{attribute addProperty BoxType "AX5021-0000-0002-0002"}
{attribute addProperty Id "Drive_status_wordAT %I*UINT162"}
{attribute addProperty CRC "4131886952"}
{attribute addProperty SizeInBites "16"}
{attribute addProperty SizeInBytes "2"}
TYPE AT_x_F6479768 :
STRUCT
	{attribute addProperty Name "Drive_status_word"}
	Drive_status_word AT %I* : UINT;
END_STRUCT
END_TYPE

(* stored: Version 1.2.0.0, ProductVersion 3.1.4024.9
   DUT AT_x_F6479768: Id {dc6497b1-a13c-4d8e-8dd8-6a4002c41d0c} *)
